{attribute 'qualified_only'}
{attribute 'strict'}
TYPE ProfileLimits :
(
	Acc0Acc1Vel,
  Vel, 
  Acc0,
  Acc1,
  Acc0Acc1,
  Acc0Vel,
  Acc1Vel,
  None
);
END_TYPE

(* stored: Version 1.1.0.1
   DUT ProfileLimits: Id {bd5b0c3f-6bf6-4746-af09-80103c0606f6} *)
